Staubli VAL3: decodeBlend.pgx

program decodeBlend(mdesc& value, num& buffer[])
  local num decodeBuffer[2]
begin
  if buffer[0] == 0
    value.blend = off
  elseIf buffer[0] == 1
    value.blend = joint
  elseIf buffer[0] == 2
    value.blend = Cartesian
  endIf

  fromBinary(buffer[1], 8, "4.0b", decodeBuffer)

  value.leave = decodeBuffer[0]
  value.reach = decodeBuffer[1]

  logMsg("B: (" + toString("", value.blend) + ", " + toString("", value.leave) + ", " + toString("", value.reach) + ")")
end
